Yaskawa INFORM job: TEA.JBI

/JOB
//NAME TEA
//POS
///NPOS 34,0,0,0
///TOOL 0
///PULSE
C000=9661,34625,-47975,4985,6680,-1354
C001=9661,33401,-46544,3989,6441,-693
C002=4571,35634,-42993,-136,3905,2448
C003=4005,39446,-40957,-488,1712,2590
C004=4582,35512,-43029,-92,4061,2429
C005=5132,32746,-43616,427,5219,2108
C006=5132,31353,-41193,357,4587,2162
C007=5177,38310,-40221,342,4332,2169
C008=4566,43109,-38146,-260,2054,2444
C009=4255,44689,-36029,-455,546,2471
C010=4814,41953,-37291,-168,2183,2384
C011=6828,41696,-37401,-118,2225,2036
C012=8409,44148,-40904,-87,3148,1774
C013=7942,45755,-39623,-471,1988,1932
C014=7647,47461,-38404,-671,1106,1976
C015=8314,44405,-40353,-214,2759,1822
C016=9442,41554,-41367,-206,3034,1637
C017=11828,41003,-41610,-174,3117,1230
C018=13380,41948,-41189,-148,3018,961
C019=12205,44745,-38610,-1199,845,1296
C020=11944,45700,-38199,-1361,438,1321
C021=13195,41949,-40173,-309,2573,1030
C022=14179,38622,-38788,354,2860,679
C023=14859,29165,-40060,401,3182,539
C024=14584,31558,-43681,-18,3787,720
C025=12953,33851,-42458,-1003,2325,1290
C026=12418,34773,-41954,-1313,1638,1413
C027=12216,35126,-41702,-1456,1292,1450
C028=11958,31225,-36746,-1866,-691,1211
C029=10405,33774,-31182,-3282,-3617,550
C030=13987,28639,-30280,-574,-341,785
C031=14204,16112,-26554,1487,1044,816
C032=9473,26781,-37799,1360,4203,1100
C033=9661,33604,-46792,4138,6486,-793
//INST
///DATE 2014/10/05 02:41
///ATTR 0,0,0,0,0,0,0,0,0,0,0,0,0,0,0,0
///FRAME BASE
NOP
*1
MOVJ C000 VJ=25.00 CONT
PAUSE
MOVJ C001 VJ=25.00 CONT
MOVJ C002 VJ=15.00 CONT
MOVJ C003 VJ=5.00 CONT
TIMER T=2.70
MOVJ C004 VJ=10.00 CONT
MOVJ C005 VJ=25.00 CONT
MOVJ C006 VJ=20.00 CONT
MOVJ C007 VJ=25.00 CONT
MOVJ C008 VJ=12.50 CONT
MOVJ C009 VJ=12.50 CONT
TIMER T=2.70
MOVJ C010 VJ=25.00 CONT
MOVJ C011 VJ=25.00 CONT
MOVJ C012 VJ=25.00 CONT
MOVJ C013 VJ=12.50 CONT
MOVJ C014 VJ=12.50 CONT
TIMER T=1.00
MOVJ C015 VJ=25.00 CONT
MOVJ C016 VJ=25.00 CONT
MOVJ C017 VJ=25.00 CONT
MOVJ C018 VJ=25.00 CONT
MOVJ C019 VJ=12.50 CONT
MOVJ C020 VJ=12.50 CONT
TIMER T=1.00
MOVJ C021 VJ=25.00 CONT
MOVJ C022 VJ=25.00 CONT
MOVJ C023 VJ=25.00 CONT
MOVJ C024 VJ=25.00 CONT
MOVJ C025 VJ=12.50 CONT
MOVJ C026 VJ=12.50 CONT
MOVJ C027 VJ=12.50 CONT
MOVJ C028 VJ=12.50 CONT
MOVJ C029 VJ=12.50 CONT
TIMER T=2.00
MOVJ C030 VJ=25.00 CONT
MOVJ C031 VJ=25.00 CONT
MOVJ C032 VJ=25.00 CONT
MOVJ C033 VJ=25.00 CONT
JUMP *1
END
